// Mitsubishi GX Works2 project: PLC   PLC: Q03UD

PROGRAM OUTPUT
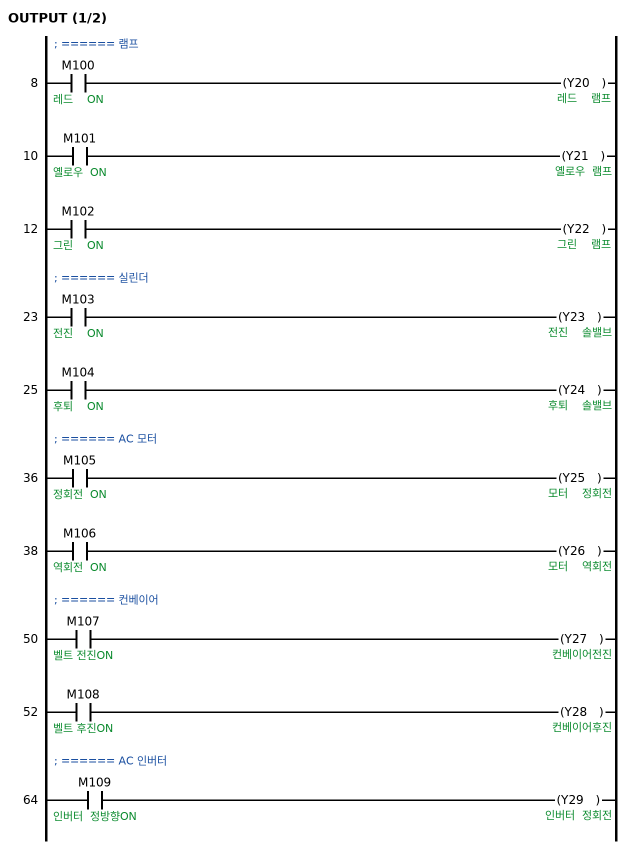
; ====== 램프
8     LD      M100  ; 레드    ON
      OUT     Y20  ; 레드    램프
10    LD      M101  ; 옐로우  ON
      OUT     Y21  ; 옐로우  램프
12    LD      M102  ; 그린    ON
      OUT     Y22  ; 그린    램프
; ====== 실린더
23    LD      M103  ; 전진    ON
      OUT     Y23  ; 전진    솔밸브
25    LD      M104  ; 후퇴    ON
      OUT     Y24  ; 후퇴    솔밸브
; ====== AC 모터
36    LD      M105  ; 정회전  ON
      OUT     Y25  ; 모터    정회전
38    LD      M106  ; 역회전  ON
      OUT     Y26  ; 모터    역회전
; ====== 컨베이어
50    LD      M107  ; 벨트 전진ON
      OUT     Y27  ; 컨베이어전진
52    LD      M108  ; 벨트 후진ON
      OUT     Y28  ; 컨베이어후진
; ====== AC 인버터
64    LD      M109  ; 인버터  정방향ON
      OUT     Y29  ; 인버터  정회전
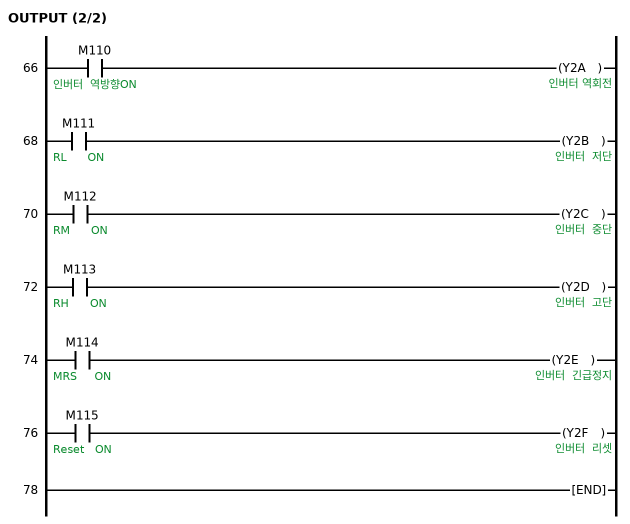
66    LD      M110  ; 인버터  역방향ON
      OUT     Y2A  ; 인버터 역회전
68    LD      M111  ; RL      ON
      OUT     Y2B  ; 인버터  저단
70    LD      M112  ; RM      ON
      OUT     Y2C  ; 인버터  중단
72    LD      M113  ; RH      ON
      OUT     Y2D  ; 인버터  고단
74    LD      M114  ; MRS     ON
      OUT     Y2E  ; 인버터  긴급정지
76    LD      M115  ; Reset   ON
      OUT     Y2F  ; 인버터  리셋
78    END
END_PROGRAM

PROGRAM INPUT
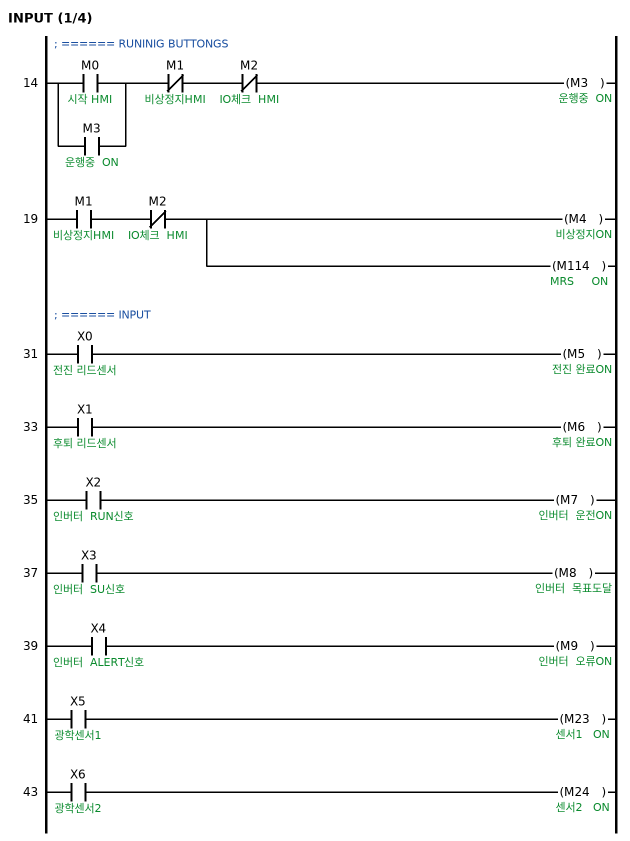
; ====== RUNINIG BUTTONGS
14    LD      M0  ; 시작 HMI
      OR      M3  ; 운행중  ON
      ANI     M1  ; 비상정지HMI
      ANI     M2  ; IO체크  HMI
      OUT     M3  ; 운행중  ON
19    LD      M1  ; 비상정지HMI
      ANI     M2  ; IO체크  HMI
      OUT     M4  ; 비상정지ON
      OUT     M114  ; MRS     ON
; ====== INPUT
31    LD      X0  ; 전진 리드센서
      OUT     M5  ; 전진 완료ON
33    LD      X1  ; 후퇴 리드센서
      OUT     M6  ; 후퇴 완료ON
35    LD      X2  ; 인버터  RUN신호
      OUT     M7  ; 인버터  운전ON
37    LD      X3  ; 인버터  SU신호
      OUT     M8  ; 인버터  목표도달
39    LD      X4  ; 인버터  ALERT신호
      OUT     M9  ; 인버터  오류ON
41    LD      X5  ; 광학센서1
      OUT     M23  ; 센서1   ON
43    LD      X6  ; 광학센서2
      OUT     M24  ; 센서2   ON
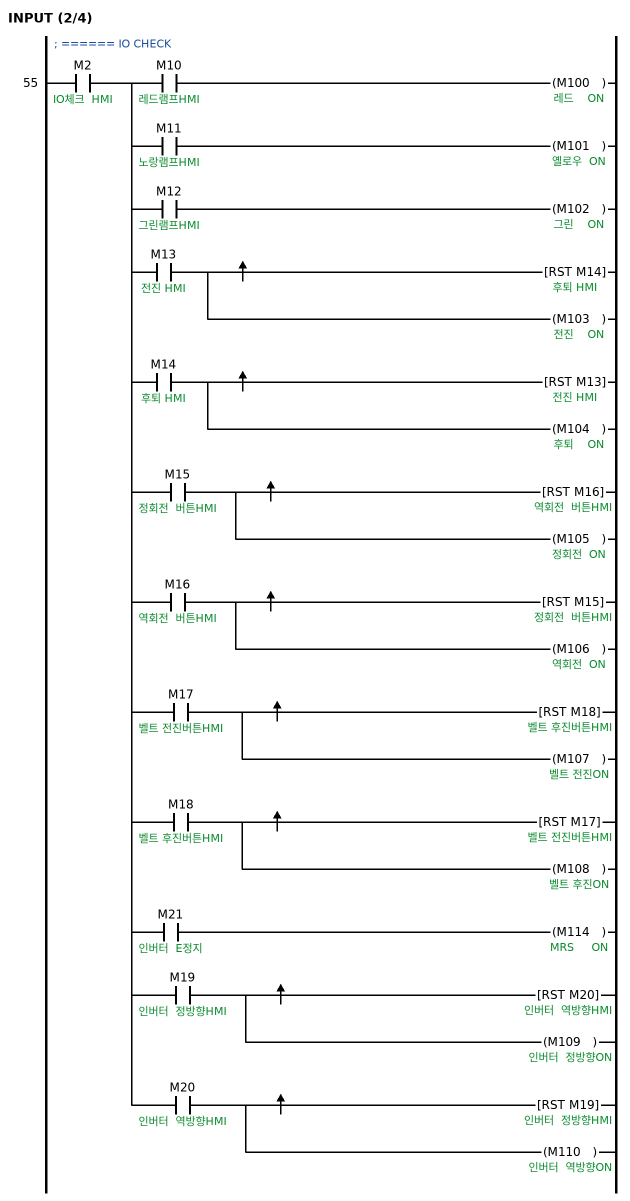
; ====== IO CHECK
55    LD      M2  ; IO체크  HMI
      MPS
      AND     M10  ; 레드램프HMI
      OUT     M100  ; 레드    ON
      MRD
      AND     M11  ; 노랑램프HMI
      OUT     M101  ; 옐로우  ON
      MRD
      AND     M12  ; 그린램프HMI
      OUT     M102  ; 그린    ON
      MRD
      AND     M13  ; 전진 HMI
      MPS
      MEP
      RST     M14  ; 후퇴 HMI
      MPP
      OUT     M103  ; 전진    ON
      MRD
      AND     M14  ; 후퇴 HMI
      MPS
      MEP
      RST     M13  ; 전진 HMI
      MPP
      OUT     M104  ; 후퇴    ON
      MRD
      AND     M15  ; 정회전  버튼HMI
      MPS
      MEP
      RST     M16  ; 역회전  버튼HMI
      MPP
      OUT     M105  ; 정회전  ON
      MRD
      AND     M16  ; 역회전  버튼HMI
      MPS
      MEP
      RST     M15  ; 정회전  버튼HMI
      MPP
      OUT     M106  ; 역회전  ON
      MRD
      AND     M17  ; 벨트 전진버튼HMI
      MPS
      MEP
      RST     M18  ; 벨트 후진버튼HMI
      MPP
      OUT     M107  ; 벨트 전진ON
      MRD
      AND     M18  ; 벨트 후진버튼HMI
      MPS
      MEP
      RST     M17  ; 벨트 전진버튼HMI
      MPP
      OUT     M108  ; 벨트 후진ON
      MRD
      AND     M21  ; 인버터  E정지
      OUT     M114  ; MRS     ON
      MRD
      AND     M19  ; 인버터  정방향HMI
      MPS
      MEP
      RST     M20  ; 인버터  역방향HMI
      MPP
      OUT     M109  ; 인버터  정방향ON
      MPP
      AND     M20  ; 인버터  역방향HMI
      MPS
      MEP
      RST     M19  ; 인버터  정방향HMI
      MPP
      OUT     M110  ; 인버터  역방향ON
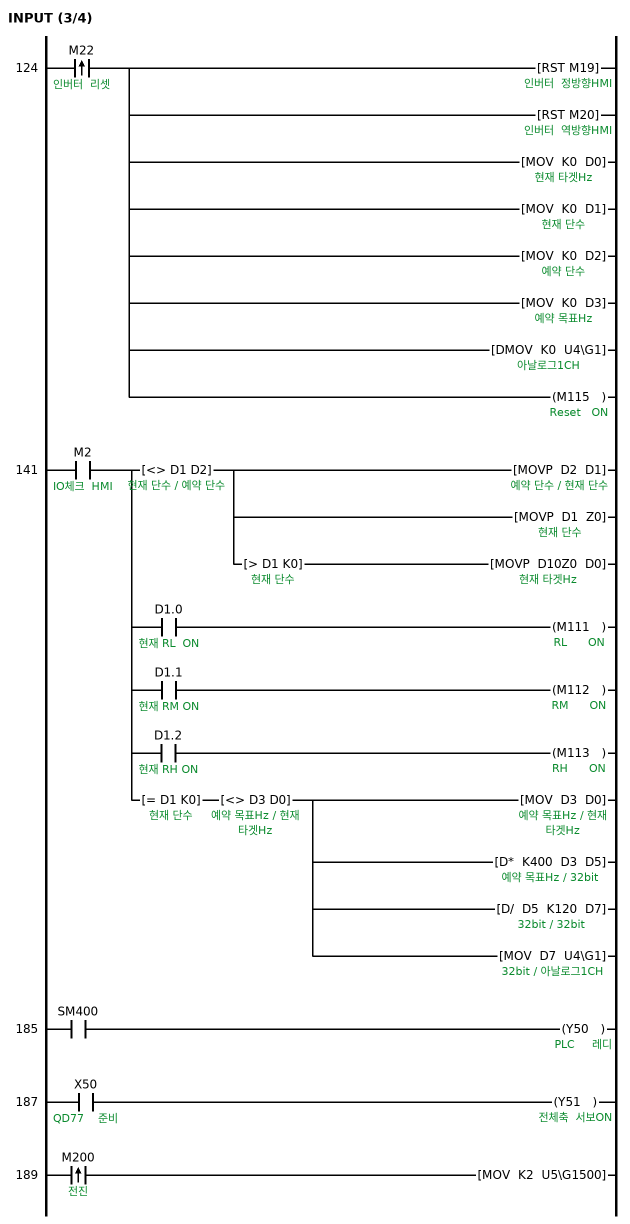
124   LDP     M22  ; 인버터  리셋
      RST     M19  ; 인버터  정방향HMI
      RST     M20  ; 인버터  역방향HMI
      MOV     K0 D0  ; 현재 타겟Hz
      MOV     K0 D1  ; 현재 단수
      MOV     K0 D2  ; 예약 단수
      MOV     K0 D3  ; 예약 목표Hz
      DMOV    K0 U4\G1  ; 아날로그1CH
      OUT     M115  ; Reset   ON
141   LD      M2  ; IO체크  HMI
      MPS
      AND<>   D1 D2  ; 현재 단수 / 예약 단수
      MOVP    D2 D1
      MOVP    D1 Z0
      AND>    D1 K0  ; 현재 단수
      MOVP    D10Z0 D0
      MRD
      AND     D1.0  ; 현재 RL  ON
      OUT     M111  ; RL      ON
      MRD
      AND     D1.1  ; 현재 RM ON
      OUT     M112  ; RM      ON
      MRD
      AND     D1.2  ; 현재 RH ON
      OUT     M113  ; RH      ON
      MPP
      AND=    D1 K0  ; 현재 단수
      AND<>   D3 D0  ; 예약 목표Hz / 현재 타겟Hz
      MOV     D3 D0
      D*      K400 D3 D5  ; 32bit
      D/      D5 K120 D7  ; 32bit
      MOV     D7 U4\G1
185   LD      SM400
      OUT     Y50  ; PLC     레디
187   LD      X50  ; QD77    준비
      OUT     Y51  ; 전체축  서보ON
189   LDP     M200  ; 전진
      MOV     K2 U5\G1500
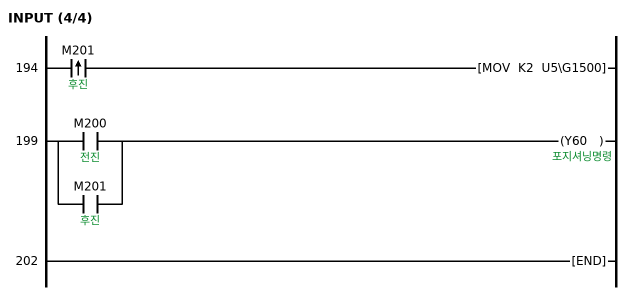
194   LDP     M201  ; 후진
      MOV     K2 U5\G1500
199   LD      M200  ; 전진
      OR      M201  ; 후진
      OUT     Y60  ; 포지셔닝명령
202   END
END_PROGRAM

PROGRAM INITIAL
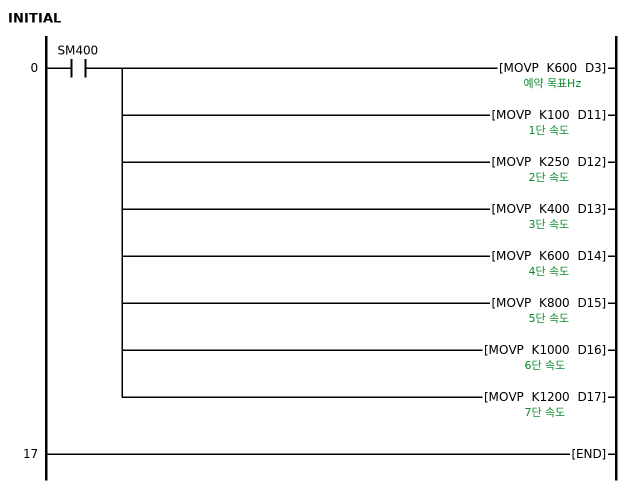
0     LD      SM400
      MOVP    K600 D3  ; 예약 목표Hz
      MOVP    K100 D11  ; 1단 속도
      MOVP    K250 D12  ; 2단 속도
      MOVP    K400 D13  ; 3단 속도
      MOVP    K600 D14  ; 4단 속도
      MOVP    K800 D15  ; 5단 속도
      MOVP    K1000 D16  ; 6단 속도
      MOVP    K1200 D17  ; 7단 속도
17    END
END_PROGRAM

// device comments not shown above
D10  ; 0단
